ABB RobotStudio station: trabajov2.rspag

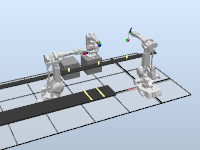
--- station ---
Station trabajov2 (saved by RobotStudio 20.4.9280.0)
Controller Controlador10, task T_ROB1: task frame (RAPID world) sits at (2700, -200, 0) mm, rotated rx 0 ry 0 rz 180 deg in the station
Controller Controlador9, task T_ROB1: task frame (RAPID world) sits at (949.84, -1514.81, 500) mm, rotated rx 0 ry 0 rz 90 deg in the station
Controller Controlador7, task T_ROB1: task frame (RAPID world) sits at (0, 250, 0) mm, rotated rx 0 ry 0 rz -90 deg in the station
Controller Controlador7
  mechanical unit ROB_1: Robot1, 6 joints, base frame (0, 0, 0) mm
Controller Controlador9
  mechanical unit ROB_1: Robot2, 6 joints, base frame (0, 0, 0) mm
Controller Controlador10
  mechanical unit ROB_1: Robot3, 6 joints, base frame (0, 0, 0) mm
Layout (positions relative to the parent item):
  - Cinta [part]
  - Botella [part]
  - Robot1 [mechanism, from Robots\IRB2400_10_150_G_02.rslib] at (0, 250, 0) mm, rotated rx 0 ry 0 rz -90 deg; joint values [0, 0.0067, 0.3043, 0, 0.3205, 0] (rad or m)
  - Llenado [mechanism, from Tools\AW_Gun_PSF_25.rslib] at (0, -678.61, 1412.5) mm, rotated rx 180 ry 60 rz 90 deg
  - SensorLlenado [smart component]
      signals: DI ActivaSensores, DO DetectadoLlenado
      connections:
        SensorLlenado.ActivaSensores -> LineSensor.Active
        LineSensor.SensorOut -> SensorLlenado.DetectadoLlenado
    - LineSensor [smart component, from Components\LineSensor.rslib] at (40, -900, 530) mm
        properties: Start=[0 0 0]; End=[0 0 0.1]; Radius=0.001; SensedPart=(none); SensedPoint=[0.04 -0.9 0.53]
      - _sensorPart_ [part]
  - CintaTransportadora [smart component]
      signals: DI NuevaBotella, DI MueveCinta, DI Desencolar, DI ParadaParaLlenar
      connections:
        CintaTransportadora.NuevaBotella -> GeneradorBotella.Execute
        GeneradorBotella.Executed -> Queue.Enqueue
        CintaTransportadora.Desencolar -> Queue.Dequeue
        CintaTransportadora.MueveCinta -> LogicGate.InputA
        CintaTransportadora.ParadaParaLlenar -> LogicGate.InputB
        CintaTransportadora.ParadaParaLlenar -> GeneradorBotella.Execute
        LogicGate_2.Output -> LogicGate_3.InputA
        LogicGate.Output -> LogicGate_3.InputB
        LogicGate_3.Output -> LinearMover.Execute
        CintaTransportadora.MueveCinta -> LogicGate_3.InputB
        CintaTransportadora.ParadaParaLlenar -> LogicGate_2.InputA
        GeneradorBotella.Copy => Queue.Back
    - LinearMover [smart component, from Components\LinearMover.rslib]
        properties: Object=Queue; Direction=[1 0 0]; Speed=0.2; Reference=Global; ReferenceObject=(none)
    - GeneradorBotella [smart component, from Components\Source.rslib]
        properties: Source=Botella; Copy=(none); Parent=(none); Position=[-0.95 -0.9 0.53]; Orientation=[0 0 0]; Transient=false; PhysicsBehavior=0
    - Queue [smart component, from Components\Queue.rslib]
        properties: Back=(none); Front=(none); Queue={48e2b2bc-c5b5-4255-99f1-ea17251d4263};{d0b61781-61f0-46d9-b633-b3a12d6bb39b}; NumberOfObjects=2
    - LogicGate_2 [smart component, from Components\LogicGate.rslib]
        properties: Operator=NOT; Delay=0
    - LogicGate_3 [smart component, from Components\LogicGate.rslib]
        properties: Operator=AND; Delay=0
  - SoporteR2 [part] at (0, -50, 0) mm
  - Robot2 [mechanism, from Robots\IRB140_6_81_C_G_03.rslib] at (949.84, -1514.81, 500) mm, rotated rx 0 ry 0 rz 90 deg; joint values [-0.2361, 0.5852, -0.3063, 0, 1.2919, -0.0099] (rad or m)
  - VentosaChapa [mechanism] at (949.84, -1008.52, 1179.5) mm, rotated rx 180 ry 60 rz -90 deg
      TCP Ventosa at (0, 0, 75) mm
      links: Pieza_12
  - SoportesChapas [part] at (-250, 0, 0) mm
  - SensorRChapa [smart component]
      signals: DO piezaDetectada, DO Vacuestato, DI ActivaVentosa, DI ActivaSensor, DO DetectadoBotellaChapa
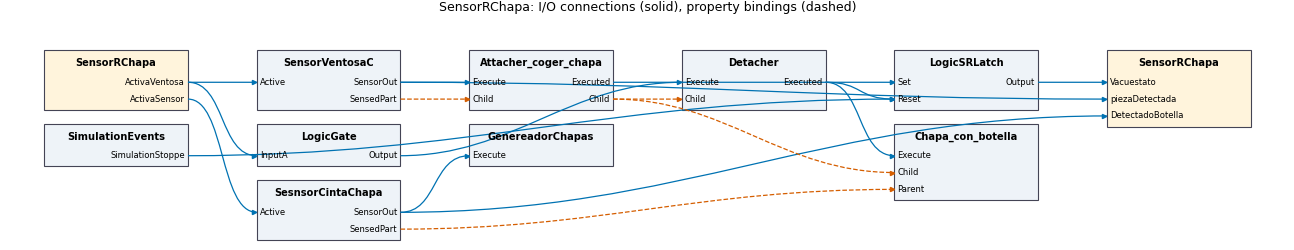
      connections:
        SensorRChapa.ActivaVentosa -> SensorVentosaC.Active
        SensorVentosaC.SensorOut -> Attacher_coger_chapa.Execute
        Attacher_coger_chapa.Executed -> LogicSRLatch.Set
        LogicSRLatch.Output -> SensorRChapa.Vacuestato
        SensorVentosaC.SensorOut -> SensorRChapa.piezaDetectada
        SensorRChapa.ActivaVentosa -> LogicGate.InputA
        LogicGate.Output -> Detacher.Execute
        Detacher.Executed -> LogicSRLatch.Reset
        SimulationEvents.SimulationStopped -> LogicSRLatch.Reset
        SensorRChapa.ActivaSensor -> SesnsorCintaChapa.Active
        SesnsorCintaChapa.SensorOut -> SensorRChapa.DetectadoBotellaChapa
        Detacher.Executed -> Chapa_con_botella.Execute
        SesnsorCintaChapa.SensorOut -> GenereadorChapas.Execute
        SensorVentosaC.SensedPart => Attacher_coger_chapa.Child
        Attacher_coger_chapa.Child => Detacher.Child
        Attacher_coger_chapa.Child => Chapa_con_botella.Child
        SesnsorCintaChapa.SensedPart => Chapa_con_botella.Parent
    - SensorVentosaC [smart component, from Components\LineSensor.rslib] at (949.84, -943.57, 1142) mm, rotated rx 180 ry 60 rz -90 deg
        properties: Start=[0 0 -0.002]; End=[0 0 0.01]; Radius=0.002; SensedPart=(none); SensedPoint=[0 0 0]
      - _sensorPart_ [part]
    - SimulationEvents [smart component, from Components\SimulationEvents.rslib]
    - LogicSRLatch [smart component, from Components\LogicSRLatch.rslib]
    - Attacher_coger_chapa [smart component, from Components\Attacher.rslib]
        properties: Parent=VentosaChapa; Flange=0; Child=(none); Mount=false; Offset=[0 0 0]; Orientation=[0 0 0]
    - Detacher [smart component, from Components\Detacher.rslib]
        properties: Child=(none); KeepPosition=true
    - LogicGate [smart component, from Components\LogicGate.rslib]
        properties: Operator=NOT; Delay=0
    - SesnsorCintaChapa [smart component, from Components\LineSensor.rslib] at (991, -900, 530) mm
        properties: Start=[0 0 0]; End=[0 0 0.1]; Radius=0.001; SensedPart=(none); SensedPoint=[0 0 0]
      - _sensorPart_ [part]
    - GenereadorChapas [smart component, from Components\Source.rslib] at (951, 0, 0) mm
        properties: Source=Chapa; Copy=(none); Parent=(none); Position=[1.678276 -1.564812 0.317]; Orientation=[0 0 0]; Transient=false; PhysicsBehavior=0
    - Chapa_con_botella [smart component, from Components\Attacher.rslib]
        properties: Parent=(none); Flange=0; Child=(none); Mount=false; Offset=[0 0 0]; Orientation=[0 0 0]
  - Chapa [part]
  - Cinta2 [part] at (0, -200, 0) mm
  - Robot3 [mechanism, from Robots\IRB2400_10_150_G_02.rslib] at (2700, -200, 0) mm, rotated rx 0 ry 0 rz 180 deg; joint values [-0.8046, 0.4446, 0.5255, 0, 1.0453, 0.7661] (rad or m)
  - CajaPequeña [part]
  - CajaGrande [part]
  - VentosaCoger [mechanism] at (1771.39, -200, 1412.5) mm, rotated rx 180 ry 60 rz 0 deg
      TCP Ventosa at (0, 0, 75) mm
      links: Pieza_12
  - CintaTransCajas [smart component]
      signals: DI CajaGrande, DI CajaPequeña, DI MoverCinta
      connections:
        NCajaPequeña.Executed -> Queue.Enqueue
        NCajaGrande.Executed -> Queue.Enqueue
        CintaTransCajas.MoverCinta -> LinearMover.Execute
        CintaTransCajas.CajaPequeña -> NCajaPequeña.Execute
        CintaTransCajas.CajaGrande -> NCajaGrande.Execute
        NCajaPequeña.Copy => Queue.Back
        NCajaGrande.Copy => Queue.Back
    - NCajaPequeña [smart component, from Components\Source.rslib] at (0, 0, 0) mm
        properties: Source=CajaPequeña; Copy=(none); Parent=(none); Position=[1.3 0.405 0.55]; Orientation=[0 0 0]; Transient=false; PhysicsBehavior=0
    - NCajaGrande [smart component, from Components\Source.rslib]
        properties: Source=CajaGrande; Copy=(none); Parent=(none); Position=[1.3 0.405 0.55]; Orientation=[0 0 0]; Transient=false; PhysicsBehavior=0
    - Queue [smart component, from Components\Queue.rslib]
        properties: Back=(none); Front=(none); Queue={9582296c-c8ea-4a8f-90e4-4259518e42be};{7a407779-05f7-4746-b3dd-5f42063eefbb};{2e4d061f-8411-411b-bf9b-926dd28ca7bb};{230ca84f-a3e5-4288-bb5b-2b5a0f1f6213};{9fdb68d5-83e2-4a01-9762-a1285b4cc58f}; NumberOfObjects=1
    - LinearMover [smart component, from Components\LinearMover.rslib]
        properties: Object=Queue; Direction=[1 0 0]; Speed=0.2; Reference=Global; ReferenceObject=(none)
  - SensorCoger [smart component]
      signals: DI Activasensor, DO DetectadoBotella, DI ActivaVentosa, DO Vacuestato, DO DetectadoCaja, DO DetectadoCajaGrande
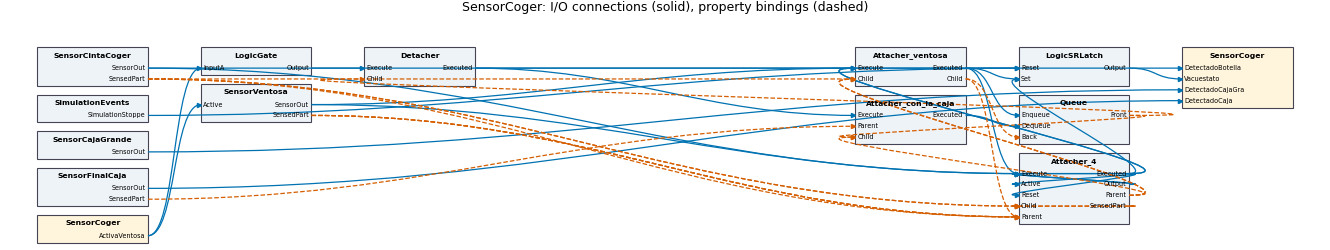
      connections:
        SensorCintaCoger.SensorOut -> SensorCoger.DetectadoBotella
        LogicGate.Output -> Detacher.Execute
        SimulationEvents.SimulationStopped -> LogicSRLatch.Reset
        Detacher.Executed -> LogicSRLatch.Reset
        LogicSRLatch.Output -> SensorCoger.Vacuestato
        SensorCajaGrande.SensorOut -> SensorCoger.DetectadoCajaGrande
        SensorFinalCaja.SensorOut -> SensorCoger.DetectadoCaja
        Detacher.Executed -> Attacher_con_la_caja.Execute
        SensorCoger.ActivaVentosa -> SensorVentosa.Active
        Attacher_4.Executed -> Attacher_ventosa.Execute
        SensorCoger.ActivaVentosa -> LogicGate.InputA
        Detacher_3.Executed -> SetParent.Execute
        Attacher_ventosa.Executed -> Attacher_5.Execute
        Attacher_5.Executed -> LogicSRLatch.Set
        Detacher_3.Executed -> Attacher_6.Execute
        Attacher_6.Executed -> Attacher_ventosa.Execute
        Attacher_ventosa.Executed -> LogicSRLatch.Set
        SensorVentosa.SensorOut -> Attacher_7.Execute
        SensorVentosa.SensorOut -> Attacher_ventosa.Execute
        SensorCintaCoger.SensorOut -> Repeater.Execute
        Repeater.Output -> Detacher_3.Execute
        Detacher_3.Executed -> Timer.Active
        Timer.Output -> Attacher_8.Execute
        Attacher_8.Executed -> Timer.Reset
        Attacher_ventosa.Executed -> Queue.Enqueue
        Attacher_con_la_caja.Executed -> Queue.Dequeue
        SensorFinalCaja.SensedPart => Attacher_con_la_caja.Parent
        SensorCintaCoger.SensedPart => SetParent.Child
        SensorVentosa.SensedPart => SetParent.Parent
        SetParent.Parent => Attacher_ventosa.Child
        Attacher_ventosa.Child => Attacher_5.Parent
        Attacher_5.Parent => Attacher_con_la_caja.Child
        SensorVentosa.SensedPart => Attacher_6.Parent
        SensorCintaCoger.SensedPart => Attacher_6.Child
        Attacher_6.Parent => Attacher_ventosa.Child
        Lineaux.SensedPart => Detacher_3.Child
        SensorVentosa.SensedPart => Attacher_7.Parent
        SensorCintaCoger.SensedPart => Attacher_8.Parent
        Lineaux.SensedPart => Attacher_8.Child
        SensorCintaCoger.SensedPart => Attacher_ventosa.Child
        Attacher_ventosa.Child => Queue.Back
        Queue.Front => Detacher.Child
        Queue.Front => Attacher_con_la_caja.Child
    - SensorCintaCoger [smart component, from Components\LineSensor.rslib]
        properties: Start=[1.9412 -0.9 0.53]; End=[1.9412 -0.9 0.63]; Radius=0.001; SensedPart=(none); SensedPoint=[0 0 0]
      - _sensorPart_ [part]
    - Attacher_ventosa [smart component, from Components\Attacher.rslib]
        properties: Parent=VentosaCoger; Flange=0; Child=(none); Mount=false; Offset=[0 0 0]; Orientation=[0 0 0]
    - LogicGate [smart component, from Components\LogicGate.rslib]
        properties: Operator=NOT; Delay=0
    - Detacher [smart component, from Components\Detacher.rslib]
        properties: Child=(none); KeepPosition=true
    - LogicSRLatch [smart component, from Components\LogicSRLatch.rslib]
    - SimulationEvents [smart component, from Components\SimulationEvents.rslib]
    - SensorFinalCaja [smart component, from Components\LineSensor.rslib]
        properties: Start=[2 0.3 0.555]; End=[2 0.8 0.555]; Radius=0.002; SensedPart=(none); SensedPoint=[2 0.405 0.555]
      - _sensorPart_ [part]
    - SensorCajaGrande [smart component, from Components\LineSensor.rslib]
        properties: Start=[1.65 0.3 0.555]; End=[1.65 0.8 0.555]; Radius=0.002; SensedPart=(none); SensedPoint=[1.65 0.405 0.555]
      - _sensorPart_ [part]
    - Attacher_con_la_caja [smart component, from Components\Attacher.rslib]
        properties: Parent=(none); Flange=0; Child=(none); Mount=false; Offset=[0 0 0]; Orientation=[0 0 0]
    - SensorVentosa [smart component, from Components\LineSensor.rslib] at (1706.44, -200, 1375) mm, rotated rx 180 ry 60 rz 0 deg
        properties: Start=[0 0 -0.002]; End=[0 0 0.02]; Radius=0.002; SensedPart=(none); SensedPoint=[0 0 0]
      - _sensorPart_ [part]
    - Queue [smart component, from Components\Queue.rslib]
        properties: Back=(none); Front=(none); Queue=; NumberOfObjects=0
  - Chapa_1 [part] at (1678.28, -1564.81, 317) mm
Attachment: SensorVentosaC is attached to VentosaChapa / Pieza_12
Attachment: NCajaPequeña is attached to Llenado / Gun
Attachment: SensorVentosa is attached to VentosaCoger / Pieza_12
Attachment: Llenado is attached to Robot1 / Link6
Attachment: VentosaChapa is attached to Robot2 / Link6
Attachment: VentosaCoger is attached to Robot3 / Link6
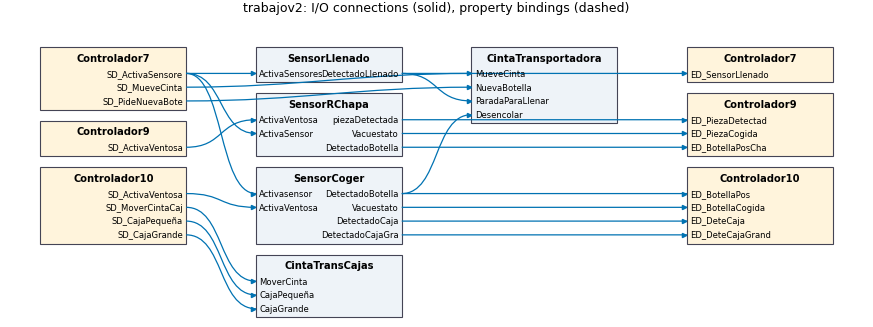
Station logic (signal -> signal, property => property):
  Controlador7.SD_ActivaSensores -> SensorLlenado.ActivaSensores
  Controlador7.SD_MueveCinta -> CintaTransportadora.MueveCinta
  Controlador7.SD_PideNuevaBotella -> CintaTransportadora.NuevaBotella
  SensorLlenado.DetectadoLlenado -> Controlador7.ED_SensorLlenado
  SensorLlenado.DetectadoLlenado -> CintaTransportadora.ParadaParaLlenar
  SensorRChapa.piezaDetectada -> Controlador9.ED_PiezaDetectada
  Controlador9.SD_ActivaVentosa -> SensorRChapa.ActivaVentosa
  SensorRChapa.Vacuestato -> Controlador9.ED_PiezaCogida
  SensorRChapa.DetectadoBotellaChapa -> Controlador9.ED_BotellaPosChapa
  SensorCoger.DetectadoBotella -> Controlador10.ED_BotellaPos
  Controlador7.SD_ActivaSensores -> SensorCoger.Activasensor
  Controlador7.SD_ActivaSensores -> SensorRChapa.ActivaSensor
  Controlador10.SD_ActivaVentosa -> SensorCoger.ActivaVentosa
  SensorCoger.Vacuestato -> Controlador10.ED_BotellaCogida
  Controlador10.SD_MoverCintaCajas -> CintaTransCajas.MoverCinta
  Controlador10.SD_CajaPequeña -> CintaTransCajas.CajaPequeña
  Controlador10.SD_CajaGrande -> CintaTransCajas.CajaGrande
  SensorCoger.DetectadoBotella -> CintaTransportadora.Desencolar
  SensorCoger.DetectadoCaja -> Controlador10.ED_DeteCaja
  SensorCoger.DetectadoCajaGrande -> Controlador10.ED_DeteCajaGrande

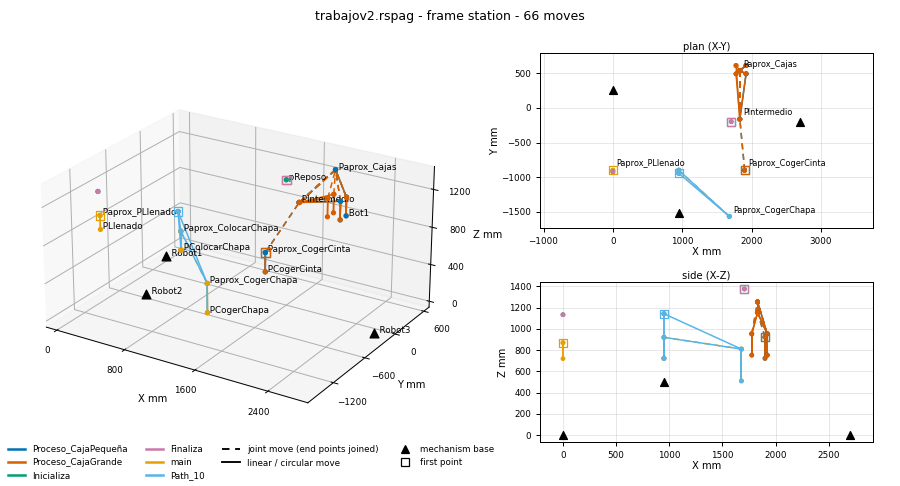
[picture p0: tool path of trabajov2.rspag in frame station, 66 of 66 moves have a stored position in this frame; points joined in program order, loops and branches not executed]
--- Backups/Controlador10/RAPID/TASK1/PROGMOD/CalibData.mod ---
MODULE CalibData
    PERS tooldata Ventosa:=[TRUE,[[0,0,75],[1,0,0,0]],[1,[0,0,20],[1,0,0,0],0,0,0]];
    TASK PERS wobjdata WCoger:=[FALSE,TRUE,"",[[0,0,0],[1,0,0,0]],[[0,0,0],[1,0,0,0]]];
ENDMODULE

--- Backups/Controlador10/RAPID/TASK1/PROGMOD/Module1.mod ---
MODULE Module1

    CONST robtarget Preposo:=[[993.564064606,0,1375],[0.5,0,0.866025404,0],[0,0,0,0],[9E+09,9E+09,9E+09,9E+09,9E+09,9E+09]];
    CONST robtarget Paprox_CogerCinta:=[[799.76,700,922.5],[0,-0.707106781,0.707106781,0],[0,0,-1,0],[9E+09,9E+09,9E+09,9E+09,9E+09,9E+09]];
    CONST robtarget PCogerCinta:=[[799.76,700,722.5],[0,-0.707106781,0.707106781,0],[0,0,-1,0],[9E+09,9E+09,9E+09,9E+09,9E+09,9E+09]];
    CONST robtarget PIntermedio:=[[869.4,-37.5,1153],[0,0.707106781,0.707106781,0],[-1,0,0,0],[9E+09,9E+09,9E+09,9E+09,9E+09,9E+09]];
    CONST robtarget Paprox_Cajas:=[[869.4,-737.5,1253],[0,0.707106781,0.707106781,0],[-1,0,0,0],[9E+09,9E+09,9E+09,9E+09,9E+09,9E+09]];
    CONST robtarget Paprox_Bot1:=[[779.4,-810,953],[0,0.707106781,0.707106781,0],[-1,0,0,0],[9E+09,9E+09,9E+09,9E+09,9E+09,9E+09]];
    CONST robtarget Bot1:=[[779.4,-810,753],[0,0.707106781,0.707106781,0],[-1,0,0,0],[9E+09,9E+09,9E+09,9E+09,9E+09,9E+09]];
    CONST robtarget Paprox_Bot2:=[[779.4,-690,953],[0,0.707106781,0.707106781,0],[-1,0,0,0],[9E+09,9E+09,9E+09,9E+09,9E+09,9E+09]];
    CONST robtarget Bot2:=[[779.4,-690,753],[0,0.707106781,0.707106781,0],[-1,0,0,0],[9E+09,9E+09,9E+09,9E+09,9E+09,9E+09]];
    CONST robtarget Paprox_Bot3G:=[[924.4,-810,953],[0,0.707106781,0.707106781,0],[-1,0,0,0],[9E+09,9E+09,9E+09,9E+09,9E+09,9E+09]];
    CONST robtarget Bot3G:=[[924.4,-810,753],[0,0.707106781,0.707106781,0],[-1,0,0,0],[9E+09,9E+09,9E+09,9E+09,9E+09,9E+09]];
    CONST robtarget Paprox_Bot4G:=[[924.4,-690,953],[0,0.707106781,0.707106781,0],[-1,0,0,0],[9E+09,9E+09,9E+09,9E+09,9E+09,9E+09]];
    CONST robtarget Bot4G:=[[924.4,-690,753],[0,0.707106781,0.707106781,0],[-1,0,0,0],[9E+09,9E+09,9E+09,9E+09,9E+09,9E+09]];
PROC main()
        Inicializa;
        SETDO SD_MoverCintaCajas,1; !Activamos el moviemiento de la cinta
        SETDO SD_CajaPequeña,1; !Creamos una caja pequeña
        SETDO SD_CajaPequeña,0;

        FOR nPiezas FROM 1 TO 10 DO ! se hace un for de 10 ya que son 20 botellas , como hay cajas de 2 lo maximo es hacerlo 10 veces(20/2=10)
        WaitDI ED_DeteCaja,1; !Esperamos que la caja este en posición
        SETDO SD_MoverCintaCajas,0;!Paramos la cinta

        IF ED_DeteCajaGrande = 0 THEN !Preguntamos si no es una caja gande
            Proceso_CajaPequeña;!Entramos en el proceso correspondiente de la caja pequeña
        ELSE
            Proceso_CajaGrande; !Entremos en el proceso correspondiente de la caja grande
        ENDIF
        ENDFOR
        Finaliza;

    ENDPROC

    PROC Proceso_CajaPequeña()
        FOR nBotellas FROM 1 TO 2 DO !se repite el for 2 veces ya que es para 2 botellas
            waitDI ED_BotellaPos,1;!Esperamos que la botella este en posicion en la cinta principal
            MoveJ Paprox_CogerCinta,v2000,fine,Ventosa\WObj:=WCoger;
            MoveL PCogerCinta,v200,fine,Ventosa\WObj:=WCoger;!Nos ponemos en poscion para cogerla
            SetDO SD_ActivaVentosa,1;!Activamos la ventosa
            WaitDI ED_BotellaCogida,1;!Esperamos el ack de que se ha cogido

            MoveL Paprox_CogerCinta,v2000,fine,Ventosa\WObj:=WCoger;
            MoveJ PIntermedio,v2000,z100,Ventosa\WObj:=WCoger;
            MoveJ Paprox_Cajas,v2000,fine,Ventosa\WObj:=WCoger;!Nos movemos al punto de aproximacion de las cajas pasando por u punto intermedio(asegurando de que no sigue un recorrido cualquiera)

            IF nBotellas = 1 THEN   !Si es la primera botella
                MoveL Paprox_Bot1,v500,fine,Ventosa\WObj:=WCoger;!Nos acermcamos al punto de aproxmiacion para colocar la botella en la pos1
                MoveL Bot1,v200,fine,Ventosa\WObj:=WCoger;
                SetDO SD_ActivaVentosa,0;
                WaitDI ED_BotellaCogida,0;!Lo soltamos
                MoveL Paprox_Bot1,v500,fine,Ventosa\WObj:=WCoger;
                MoveJ Paprox_Cajas,v2000,z100,Ventosa\WObj:=WCoger;
                MoveJ PIntermedio,v2000,z100,Ventosa\WObj:=WCoger;  !Volvenos al punto intermedio pasando por los puntos correspondiente de vuelta
            ELSE!Entramos cuando es la segunda botella, el proceso es igual que para la anterior pero cambiando los puntos de coordenadas
                MoveL Paprox_Bot2,v500,fine,Ventosa\WObj:=WCoger;
                MoveL Bot2,v200,fine,Ventosa\WObj:=WCoger;
                SetDO SD_ActivaVentosa,0;
                WaitDI ED_BotellaCogida,0;
                MoveL Paprox_Bot2,v500,fine,Ventosa\WObj:=WCoger;
            ENDIF
        ENDFOR
        SETDO SD_MoverCintaCajas,1;!una vez se han puesto todas las botellas en la caja, se activa el movimento de la cinta
        MoveJ Paprox_Cajas,v2000,z100,Ventosa\WObj:=WCoger;
        MoveJ PIntermedio,v2000,z100,Ventosa\WObj:=WCoger; !hacemos que el robot vuelva tambien al punto intermedio
        WaitDI ED_DeteCaja,0; ! Esperamos que la caja pase para crear una nueva
        SETDO SD_CajaGrande,1;!creamos una caja grande
        SETDO SD_CajaGrande,0;
    ENDPROC

    PROC Proceso_CajaGrande()   !Este proceso es igual que el de la caja pequeña pero teniendo en cuentas mas puntos para colocar las botellas por lo que el for es de 4
        FOR nBotellas FROM 1 TO 4 DO
            waitDI ED_BotellaPos,1;
            MoveJ Paprox_CogerCinta,v2000,fine,Ventosa\WObj:=WCoger;
            MoveL PCogerCinta,v200,fine,Ventosa\WObj:=WCoger;
            SetDO SD_ActivaVentosa,1;
            WaitDI ED_BotellaCogida,1;

            MoveL Paprox_CogerCinta,v2000,fine,Ventosa\WObj:=WCoger;
            MoveJ PIntermedio,v2000,z100,Ventosa\WObj:=WCoger;
            MoveJ Paprox_Cajas,v2000,fine,Ventosa\WObj:=WCoger;

            IF nBotellas = 1 THEN
                MoveL Paprox_Bot1,v500,fine,Ventosa\WObj:=WCoger;
                MoveL Bot1,v200,fine,Ventosa\WObj:=WCoger;
                SetDO SD_ActivaVentosa,0;
                WaitDI ED_BotellaCogida,0;
                MoveL Paprox_Bot1,v500,fine,Ventosa\WObj:=WCoger;
                MoveJ Paprox_Cajas,v2000,z100,Ventosa\WObj:=WCoger;
                MoveJ PIntermedio,v2000,z100,Ventosa\WObj:=WCoger;
            ELSEIF nBotellas = 2 THEN
                MoveL Paprox_Bot2,v500,fine,Ventosa\WObj:=WCoger;
                MoveL Bot2,v200,fine,Ventosa\WObj:=WCoger;
                SetDO SD_ActivaVentosa,0;
                WaitDI ED_BotellaCogida,0;
                MoveL Paprox_Bot2,v500,fine,Ventosa\WObj:=WCoger;
                MoveJ Paprox_Cajas,v2000,z100,Ventosa\WObj:=WCoger;
                MoveJ PIntermedio,v2000,z100,Ventosa\WObj:=WCoger;
            ELSEIF nBotellas = 3 THEN
                MoveL Paprox_Bot3G,v500,fine,Ventosa\WObj:=WCoger;
                MoveL Bot3G,v200,fine,Ventosa\WObj:=WCoger;
                SetDO SD_ActivaVentosa,0;
                WaitDI ED_BotellaCogida,0;
                MoveL Paprox_Bot3G,v500,fine,Ventosa\WObj:=WCoger;
                MoveJ Paprox_Cajas,v2000,z100,Ventosa\WObj:=WCoger;
                MoveJ PIntermedio,v2000,z100,Ventosa\WObj:=WCoger;
            ELSE
                MoveL Paprox_Bot4G,v500,fine,Ventosa\WObj:=WCoger;
                MoveL Bot4G,v200,fine,Ventosa\WObj:=WCoger;
                SetDO SD_ActivaVentosa,0;
                WaitDI ED_BotellaCogida,0;
                MoveL Paprox_Bot4G,v500,fine,Ventosa\WObj:=WCoger;
            ENDIF
        ENDFOR
        SETDO SD_MoverCintaCajas,1;
        MoveJ Paprox_Cajas,v2000,z100,Ventosa\WObj:=WCoger;
        MoveJ PIntermedio,v2000,z100,Ventosa\WObj:=WCoger;
        WaitDI ED_DeteCaja,0; ! ha pasado la caja
        SETDO SD_CajaPequeña,1;
        SETDO SD_CajaPequeña,0;
    ENDPROC

    PROC Inicializa ()
      MoveJ pReposo, v3000, fine,Ventosa\WObj:=wobj0;
      Reset SD_ActivaVentosa;
      Reset SD_MoverCintaCajas;
      Reset SD_CajaGrande;
      Reset SD_CajaPequeña;

   ENDPROC

   PROC Finaliza ()
      MoveJ pReposo, v3000, fine, Ventosa\WObj:=wobj0;
      Reset SD_ActivaVentosa;
      Reset SD_MoverCintaCajas;
      Reset SD_CajaGrande;
      Reset SD_CajaPequeña;
   ENDPROC

ENDMODULE

--- Backups/Controlador7/RAPID/TASK1/PROGMOD/CalibData.mod ---
MODULE CalibData
    PERS tooldata AW_Gun:=[TRUE,[[119.5,0,352],[0.890214,0,0.455543,0]],[1,[0,0,100],[1,0,0,0],0,0,0]];
    TASK PERS wobjdata W_Llenado:=[FALSE,TRUE,"",[[0,0,0],[1,0,0,0]],[[0,0,0],[1,0,0,0]]];
ENDMODULE

--- Backups/Controlador7/RAPID/TASK1/PROGMOD/Module1.mod ---
MODULE Module1

    CONST robtarget pReposo:=[[1173.703101454,0,1133.009964248],[0.050594996,0,0.998719253,0],[0,0,0,0],[9E+09,9E+09,9E+09,9E+09,9E+09,9E+09]];
    CONST robtarget Paprox_PLlenado:=[[1150,0,870],[0,0,1,0],[0,0,0,0],[9E+09,9E+09,9E+09,9E+09,9E+09,9E+09]];
    CONST robtarget PLlenado:=[[1150,0,720],[0,0,1,0],[0,0,0,0],[9E+09,9E+09,9E+09,9E+09,9E+09,9E+09]];
PROC main()


      Inicializa;

      FOR nPiezas FROM 1 TO 20 DO
         WaitDI ED_SensorLlenado, 1; !Esperamos que la botella esté en posición
         MoveL Paprox_PLlenado,v1000,z100,AW_Gun\WObj:=W_Llenado;
         MoveL PLlenado,v1000,fine,AW_Gun\WObj:=W_Llenado;
         WaitTime 3;  !3 segundos de parada simulando que se esta llenando la botella
         MoveL Paprox_PLlenado,v1000,z100,AW_Gun\WObj:=W_Llenado;
         SetDO SD_ActivaSensores, 0; !Desactivamos los sensores para que la cinta se mueva
         WaitTime 3;   !esperamos 3 segundos
         SetDO SD_ActivaSensores, 1; !volvemos a activar los sensores
      ENDFOR

      Finaliza;
    ENDPROC

    PROC Inicializa ()
      MoveJ pReposo, v3000, fine,AW_Gun\WObj:=wobj0;
      SetDO SD_ActivaSensores, 0;
      SetDO SD_MueveCinta, 1;
      SetDO SD_PideNuevaBotella,1;!Creamos una botella nueva en la cinta
      Reset SD_PideNuevaBotella;
      SetDO SD_ActivaSensores, 1; !Activamos los sensores
   ENDPROC

   PROC Finaliza ()
      MoveJ pReposo, v3000, fine, AW_Gun\WObj:=wobj0;
      Reset SD_PideNuevaBotella;
      Reset SD_MueveCinta;
      Reset SD_ActivaSensores;
   ENDPROC

ENDMODULE

--- Backups/Controlador9/RAPID/TASK1/PROGMOD/CalibData.mod ---
MODULE CalibData
    PERS tooldata Ventosa:=[TRUE,[[0,0,75],[1,0,0,0]],[1,[0,0,20],[1,0,0,0],0,0,0]];
    TASK PERS wobjdata W_Chapa:=[FALSE,TRUE,"",[[0,0,0],[1,0,0,0]],[[0,0,0],[1,0,0,0]]];
ENDMODULE

--- Backups/Controlador9/RAPID/TASK1/PROGMOD/Module1.mod ---
MODULE Module1
    CONST robtarget PReposo:=[[571.24355653,0,642],[0.5,0,0.866025404,0],[0,0,0,0],[9E+09,9E+09,9E+09,9E+09,9E+09,9E+09]];
    CONST robtarget Paprox_CogerChapa:=[[-50,-728.436,310],[0,0.707106781,0.707106781,0],[-2,0,-1,0],[9E+09,9E+09,9E+09,9E+09,9E+09,9E+09]];
    CONST robtarget PCogerChapa:=[[-50,-728.436,10],[0,0.707106781,0.707106781,0],[-2,0,-1,0],[9E+09,9E+09,9E+09,9E+09,9E+09,9E+09]];
    CONST robtarget Paprox_ColocarChapa:=[[614.812,0,420],[0,0,1,0],[0,0,0,0],[9E+09,9E+09,9E+09,9E+09,9E+09,9E+09]];
    CONST robtarget PColocarChapa:=[[614.812,0,222.5],[0,0,1,0],[0,0,0,0],[9E+09,9E+09,9E+09,9E+09,9E+09,9E+09]];
    CONST robtarget PColocarChapa_girar:=[[614.812,0,222.5],[0,0.675590207,0.737277337,0],[0,0,0,0],[9E+09,9E+09,9E+09,9E+09,9E+09,9E+09]];

PROC main()


      Inicializa;

      FOR nPiezas FROM 1 TO 20 DO
        !Lo primero que hacemos es coger la chapa
         MoveJ Paprox_CogerChapa,v1000,z100,Ventosa\WObj:=W_Chapa;
         MoveL PCogerChapa,v500,fine,Ventosa\WObj:=W_Chapa;
         SetDO SD_ActivaVentosa,1;
         WaitDI ED_PiezaCogida,1;

         !Una vez cogida la chapa nos ponemos en la posicion de aproxmacion para ponerla
         MoveL Paprox_CogerChapa,v1000,z100,Ventosa\WObj:=W_Chapa;
         MoveJ Paprox_ColocarChapa,v1000,z100,Ventosa\WObj:=W_Chapa;
         WaitDI ED_BotellaPosChapa,1;!esperamos que la botella este en posición(en este momento aparece una chapa nueva)

         MoveL PColocarChapa,v200,fine,Ventosa\WObj:=W_Chapa;!Una vez en posición colocamos la chapa
         MoveL PColocarChapa_girar,v200,fine,Ventosa\WObj:=W_Chapa;!se realiza un giro simulando ser la rosca

         SetDO SD_ActivaVentosa,0;!desactivamos la ventosa
         WaitDI ED_PiezaCogida,0;

        MoveL PColocarChapa,v200,fine,Ventosa\WObj:=W_Chapa;!volvemos a la posicion de aprox
         MoveL Paprox_ColocarChapa,v200,fine,Ventosa\WObj:=W_Chapa;

      ENDFOR

      Finaliza;
    ENDPROC

    PROC Inicializa ()
      MoveJ pReposo, v1000, fine,Ventosa\WObj:=wobj0;
      Reset SD_ActivaVentosa;

   ENDPROC

   PROC Finaliza ()
      MoveJ pReposo, v3000, fine, Ventosa\WObj:=wobj0;
      Reset SD_ActivaVentosa;
   ENDPROC

    PROC Path_10()
        MoveL PReposo,v1000,z100,Ventosa\WObj:=wobj0;
        MoveL Paprox_CogerChapa,v1000,z100,Ventosa\WObj:=W_Chapa;
        MoveL PCogerChapa,v1000,z100,Ventosa\WObj:=W_Chapa;
        MoveL Paprox_CogerChapa,v1000,z100,Ventosa\WObj:=W_Chapa;
        MoveL Paprox_ColocarChapa,v1000,z100,Ventosa\WObj:=W_Chapa;
        MoveL PColocarChapa,v1000,z100,Ventosa\WObj:=W_Chapa;
        MoveL Paprox_ColocarChapa,v1000,z100,Ventosa\WObj:=W_Chapa;
        MoveL PReposo,v1000,z100,Ventosa\WObj:=wobj0;
        MoveL PColocarChapa_girar,v1000,z100,Ventosa\WObj:=W_Chapa;
    ENDPROC

ENDMODULE

--- Backups/Controlador10/SYSPAR/EIO.cfg ---
EIO:CFG_1.0:6:1::
#
INDUSTRIAL_NETWORK:

      -Name "DeviceNet" -Label "DeviceNet Master/Slave Network" -Address "2"
#
DEVICENET_DEVICE:

      -Name "MiDeviceNet" -Label "MiDeviceNet"
#
DEVICENET_INTERNAL_DEVICE:

      -Name "DN_Internal_Device" -VendorName "ABB Robotics"\
      -ProductName "DeviceNet Internal Slave Device"
#
EIO_SIGNAL:

      -Name "SD_MoverCintaCajas" -SignalType "DO" -Device "MiDeviceNet"\
      -Label "SD_MoverCintaCajas" -DeviceMap "0" -Access "All"

      -Name "SD_CajaPequeña" -SignalType "DO" -Device "MiDeviceNet"\
      -Label "SD_CajaPequeña" -DeviceMap "1" -Access "All"

      -Name "SD_CajaGrande" -SignalType "DO" -Device "MiDeviceNet"\
      -Label "SD_CajaGrande" -DeviceMap "2" -Access "All"

      -Name "ED_BotellaPos" -SignalType "DI" -Device "MiDeviceNet"\
      -Label "ED_BotellaPos" -DeviceMap "0"

      -Name "ED_BotellaCogida" -SignalType "DI" -Device "MiDeviceNet"\
      -Label "ED_BotellaCogida" -DeviceMap "1"

      -Name "SD_ActivaVentosa" -SignalType "DO" -Device "MiDeviceNet"\
      -Label "SD_ActivaVentosa" -DeviceMap "3"

      -Name "ED_DeteCaja" -SignalType "DI" -Device "MiDeviceNet"\
      -Label "ED_DeteCaja" -DeviceMap "2"

      -Name "ED_DeteCajaGrande" -SignalType "DI" -Device "MiDeviceNet"\
      -Label "ED_DeteCajaGrande" -DeviceMap "3"

--- Backups/Controlador7/SYSPAR/EIO.cfg ---
EIO:CFG_1.0:6:1::
#
INDUSTRIAL_NETWORK:

      -Name "DeviceNet" -Label "DeviceNet Master/Slave Network" -Address "2"
#
DEVICENET_DEVICE:

      -Name "MiDeviceNet" -Label "MiDeviceNet"
#
DEVICENET_INTERNAL_DEVICE:

      -Name "DN_Internal_Device" -VendorName "ABB Robotics"\
      -ProductName "DeviceNet Internal Slave Device"
#
EIO_SIGNAL:

      -Name "ED_SensorLlenado" -SignalType "DI" -Device "MiDeviceNet"\
      -Label "ED_SensorLlenado" -DeviceMap "0" -Access "All"

      -Name "SD_ActivaSensores" -SignalType "DO" -Device "MiDeviceNet"\
      -Label "SD_ActivaSensores" -DeviceMap "0" -Access "All"

      -Name "SD_MueveCinta" -SignalType "DO" -Device "MiDeviceNet"\
      -Label "SD_MueveCinta" -DeviceMap "1" -Access "All"

      -Name "SD_PideNuevaBotella" -SignalType "DO" -Device "MiDeviceNet"\
      -Label "SD_PideNuevaBotella" -DeviceMap "3" -Access "All"

--- Backups/Controlador9/SYSPAR/EIO.cfg ---
EIO:CFG_1.0:6:1::
#
INDUSTRIAL_NETWORK:

      -Name "DeviceNet" -Label "DeviceNet Master/Slave Network" -Address "2"
#
DEVICENET_DEVICE:

      -Name "MiDeviceNet" -Label "MiDeviceNet"
#
DEVICENET_INTERNAL_DEVICE:

      -Name "DN_Internal_Device" -VendorName "ABB Robotics"\
      -ProductName "DeviceNet Internal Slave Device"
#
EIO_SIGNAL:

      -Name "ED_PiezaDetectada" -SignalType "DI" -Device "MiDeviceNet"\
      -Label "ED_PiezaDetectada" -DeviceMap "0" -Access "All"

      -Name "ED_PiezaCogida" -SignalType "DI" -Device "MiDeviceNet"\
      -Label "ED_PiezaCogida" -DeviceMap "1" -Access "All"

      -Name "SD_ActivaVentosa" -SignalType "DO" -Device "MiDeviceNet"\
      -Label "SD_ActivaVentosa" -DeviceMap "0" -Access "All"

      -Name "ED_BotellaPosChapa" -SignalType "DI" -Device "MiDeviceNet"\
      -Label "ED_BotellaPosChapa" -DeviceMap "2" -Access "All"
